// TIA Portal project "自动组装流水线" (V16)

(* hardware
DEVICE "HMI_1"  KTP700 Basic PN
   slot 0: "HMI_1"  KTP700 Basic PN  6AV2 123-2GB03-0AX0  16.0.0.0
   slot 1: "HMI_RT_1"  KTP700 Basic PN  6AV2 123-2GB03-0AX0  16.0.0.0
   slot 5: "HMI_1.IE_CP_1"  PROFINET Interface  16.0.0.0
      slot 1: "PROFINET Interface_1"  PROFINET Interface
         slot 1: "Port_1"  Port
DEVICE "S7-1200 station_1"  S7-1200 Station
   slot 0: "Rack_0"  S7-1200 Rack  Rack  V1.0
   slot 1: "PLC_1"  CPU 1214C DC/DC/Rly  6ES7 214-1HG40-0XB0  V4.4
*)

// ===== PLC "PLC_1"  CPU 1214C DC/DC/Rly =====

VAR_GLOBAL   // PLC tag table "中间变量"
   "中间变量1" AT %M0.0 : Bool;
   "中间变量2" AT %M0.1 : Bool;
   "中间变量3" AT %M0.2 : Bool;
   "中间变量4" AT %M0.3 : Bool;
   "中间变量5" AT %M0.4 : Bool;
   "中间变量6" AT %M0.5 : Bool;
   "中间变量7" AT %M0.6 : Bool;
   "中间变量8" AT %M0.7 : Bool;
   "中间变量9" AT %M1.0 : Bool;
   "中间变量10" AT %M1.1 : Bool;
   "中间变量11" AT %M1.2 : Bool;
   "中间变量12" AT %M1.3 : Bool;
   "中间变量13" AT %M1.4 : Bool;
   "中间变量14" AT %M1.5 : Bool;
   "启动" AT %M1.6 : Bool;
   "停止(1)" AT %M1.7 : Bool;
   "复位(1)" AT %M2.0 : Bool;
   "启动标志1" AT %M2.1 : Bool;
   "推杆标志1" AT %M2.2 : Bool;
   "推杆标志2" AT %M2.3 : Bool;
   "推杆收1" AT %M2.4 : Bool;
   "推杆收2" AT %M2.5 : Bool;
   "上下准备" AT %M2.6 : Bool;
   "吸附准备" AT %M2.7 : Bool;
   "吸附过程" AT %M3.0 : Bool;
   "前后准备" AT %M3.1 : Bool;
   "准备下降" AT %M3.2 : Bool;
   "断开吸附" AT %M3.3 : Bool;
   "x轴复位" AT %M3.4 : Bool;
   "皮带1状态" AT %M3.5 : Bool;
   "皮带2状态" AT %M3.6 : Bool;
   "皮带启动1" AT %M3.7 : Bool;
   "皮带启动2" AT %M4.0 : Bool;
   "上升2准备" AT %M4.1 : Bool;
   "上升2复位" AT %M4.2 : Bool;
END_VAR

VAR_GLOBAL   // PLC tag table "io表"
   "传感器9" AT %I0.0 : Bool;
   "传感器8" AT %I0.1 : Bool;
   "传感器7" AT %I0.2 : Bool;
   "传感器1" AT %I0.3 : Bool;
   "传感器2" AT %I0.4 : Bool;
   "传感器3" AT %I0.5 : Bool;
   "传感器4" AT %I0.6 : Bool;
   "传感器5" AT %I0.7 : Bool;
   "传感器6" AT %I1.0 : Bool;
   "传感器10" AT %I1.1 : Bool;
   "开始" AT %I1.2 : Bool;
   "复位" AT %I1.3 : Bool;
   "停止" AT %I1.4 : Bool;
   "紧急停止" AT %I1.5 : Bool;
   "1挡" AT %I1.6 : Bool;
   "FACTORY I/O (Running)" AT %I1.7 : Bool;
   "前后" AT %Q0.0 : Bool;
   "上下" AT %Q0.1 : Bool;
   "吸取" AT %Q0.2 : Bool;
   "皮带1" AT %Q0.3 : Bool;
   "推上盖" AT %Q0.4 : Bool;
   "上升1" AT %Q0.5 : Bool;
   "皮带2" AT %Q0.6 : Bool;
   "推下盖" AT %Q0.7 : Bool;
   "上升2" AT %Q1.0 : Bool;
   "绿灯" AT %Q1.1 : Bool;
   "黄灯" AT %Q1.2 : Bool;
   "红灯" AT %Q1.3 : Bool;
   "显示屏" AT %QD30 : DInt;
END_VAR

DATA_BLOCK "主程序"   // DB13
{ S7_Optimized_Access := 'TRUE' }
VERSION : 0.1
   VAR
      急停 : Bool := true;
      模式 : Int;
      "运行/停止" : Bool;
   END_VAR
BEGIN
END_DATA_BLOCK

// folder: 01-自动运行组装

DATA_BLOCK "自动运行组装_DB"   // DB14
{ S7_Optimized_Access := 'TRUE' }
VERSION : 0.1
// stored: InstanceOfName 自动运行组装
"自动运行组装"
BEGIN
END_DATA_BLOCK

// folder: 02-系统停止组块

DATA_BLOCK "系统停止组块_DB"   // DB2
{ S7_Optimized_Access := 'TRUE' }
VERSION : 0.1
// stored: InstanceOfName 系统停止组块
"系统停止组块"
BEGIN
END_DATA_BLOCK

// folder: System blocks/Program resources

DATA_BLOCK "IEC_Timer_0_DB_11"   // DB12
{ S7_Optimized_Access := 'TRUE' }
AUTHOR : Simatic
FAMILY : IEC
NAME : IEC_TMR
VERSION : 1.0
// stored: InstanceOfName IEC_TIMER
"IEC_TIMER"
BEGIN
END_DATA_BLOCK

// folder: (top level)

FUNCTION "MHJ-PLC-Lab-Function-S71200" : Void   // FC9000, SCL
{ S7_Optimized_Access := 'TRUE' }
VERSION : 0.1
   VAR_TEMP
      rdTimeReturn : Int;
      outputTime : DTL;
      SyncVal : Byte;
      forVal : Int;
      forVal_2 : Int;
      Value : Byte;
   END_VAR
   VAR CONSTANT
      CompVal : Byte := 16#34;
      Value_01 : Byte := 16#11;
      Value_01_DW : DWord := 16#A165_D992;
      Value_02_DW : DWord := 16#58BE_4401;
   END_VAR
BEGIN

   #Value:=PEEK(area := 16#82,
        dbNumber := 0,
        byteOffset := 511);
   #Value := #Value + 1;

   POKE(area := 16#82,
        dbNumber := 0,
        byteOffset := 511,
        value := #Value);

   POKE(area:=16#81,
        dbNumber:=0,
        byteOffset:=1016,
        value:=#Value_01_DW);
   POKE(area := 16#81,
        dbNumber := 0,
        byteOffset := 1020,
        value := #Value_02_DW);

   POKE(area := 16#81,
        dbNumber := 0,
        byteOffset := 511,
        value := B#16#00);

   FOR #forVal := 0 TO 120 DO
       FOR #forVal_2:=0 TO 10 DO
           #rdTimeReturn:=RD_SYS_T(#outputTime);
           #rdTimeReturn := WR_SYS_T(#outputTime);
           #rdTimeReturn := RD_SYS_T(#outputTime);
           #rdTimeReturn := WR_SYS_T(#outputTime);
       END_FOR;
       #SyncVal:= PEEK(area := 16#81,
                      dbNumber := 0,
                      byteOffset := 511);
       IF #SyncVal = #CompVal THEN
          GOTO M_1;
       END_IF;
   END_FOR;
   RETURN;

   M_1:
   POKE(area := 16#81,
        dbNumber := 0,
        byteOffset := 511,
        value := B#16#0);
END_FUNCTION

ORGANIZATION_BLOCK "Main"   // OB1, LAD, ProgramCycle
TITLE = "Main Program Sweep (Cycle)"
{ S7_Optimized_Access := 'TRUE' }
VERSION : 0.1
   VAR_INPUT
      Initial_Call : Bool;   // Initial call of this OB
      Remanence : Bool;   // =True, if remanent data are available
   END_VAR
   VAR_TEMP   // added for the SCL form of the ladder/FBD networks
      _w1 : Bool;
      _w2 : Bool;
   END_VAR
BEGIN

REGION Network 1
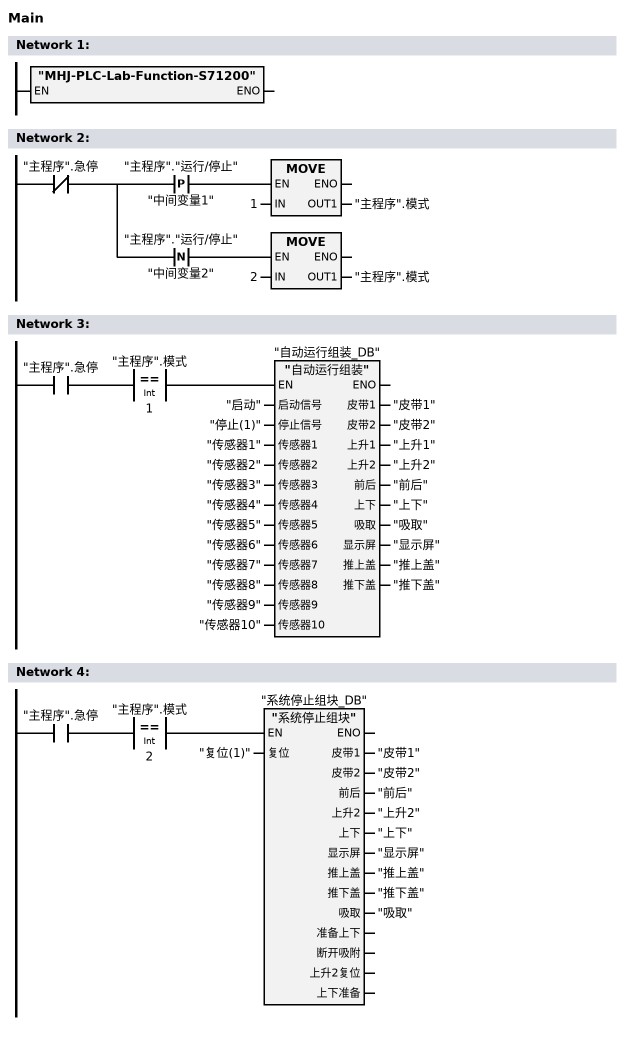
   RUNG wire#powerrail
      "MHJ-PLC-Lab-Function-S71200"()
   END_RUNG
   // the same network as SCL:
   "MHJ-PLC-Lab-Function-S71200"();
END_REGION

REGION Network 2
   RUNG wire#powerrail
      I_Contact( "主程序".急停 )
      wire#w1
      P_Contact(operand := "主程序"."运行/停止", bit := "中间变量1")
      Move(in := 1, out1 => "主程序".模式)
   END_RUNG
   RUNG wire#w1
      N_Contact(operand := "主程序"."运行/停止", bit := "中间变量2")
      Move(in := 2, out1 => "主程序".模式)
   END_RUNG
   // the same network as SCL:
   #_w1 := NOT "主程序".急停 AND "主程序"."运行/停止" AND NOT "中间变量1";   // rising edge of "主程序"."运行/停止"
   "中间变量1" := "主程序"."运行/停止";
   IF #_w1 THEN "主程序".模式 := 1; END_IF;
   #_w2 := NOT "主程序".急停 AND NOT "主程序"."运行/停止" AND "中间变量2";   // falling edge of "主程序"."运行/停止"
   "中间变量2" := "主程序"."运行/停止";
   IF #_w2 THEN "主程序".模式 := 2; END_IF;
END_REGION

REGION Network 3
   RUNG wire#powerrail
      Contact( "主程序".急停 )
      { S7_Templates := "SrcType := Int" } EQ_Contact(in1 := "主程序".模式, in2 := 1)
      "自动运行组装_DB"(启动信号 := "启动", 停止信号 := "停止(1)", 传感器1 := "传感器1", 传感器2 := "传感器2", 传感器3 := "传感器3", 传感器4 := "传感器4", 传感器5 := "传感器5", 传感器6 := "传感器6", 传感器7 := "传感器7", 传感器8 := "传感器8", 传感器9 := "传感器9", 传感器10 := "传感器10", 皮带1 => "皮带1", 皮带2 => "皮带2", 上升1 => "上升1", 上升2 => "上升2", 前后 => "前后", 上下 => "上下", 吸取 => "吸取", 显示屏 => "显示屏", 推上盖 => "推上盖", 推下盖 => "推下盖")
   END_RUNG
   // the same network as SCL:
   IF "主程序".急停 AND ("主程序".模式 = 1) THEN
       "自动运行组装_DB"(启动信号 := "启动",   // "自动运行组装"
                   停止信号 := "停止(1)",
                   传感器1 := "传感器1",
                   传感器2 := "传感器2",
                   传感器3 := "传感器3",
                   传感器4 := "传感器4",
                   传感器5 := "传感器5",
                   传感器6 := "传感器6",
                   传感器7 := "传感器7",
                   传感器8 := "传感器8",
                   传感器9 := "传感器9",
                   传感器10 := "传感器10",
                   皮带1 => "皮带1",
                   皮带2 => "皮带2",
                   上升1 => "上升1",
                   上升2 => "上升2",
                   前后 => "前后",
                   上下 => "上下",
                   吸取 => "吸取",
                   显示屏 => "显示屏",
                   推上盖 => "推上盖",
                   推下盖 => "推下盖");
   END_IF;
END_REGION

REGION Network 4
   RUNG wire#powerrail
      Contact( "主程序".急停 )
      { S7_Templates := "SrcType := Int" } EQ_Contact(in1 := "主程序".模式, in2 := 2)
      "系统停止组块_DB"(复位 := "复位(1)", 皮带1 => "皮带1", 皮带2 => "皮带2", 前后 => "前后", 上升2 => "上升2", 上下 => "上下", 显示屏 => "显示屏", 推上盖 => "推上盖", 推下盖 => "推下盖", 吸取 => "吸取", 准备上下 =>, 断开吸附 =>, 上升2复位 =>, 上下准备 =>)
   END_RUNG
   // the same network as SCL:
   IF "主程序".急停 AND ("主程序".模式 = 2) THEN
       "系统停止组块_DB"(复位 := "复位(1)",   // "系统停止组块"
                   皮带1 => "皮带1",
                   皮带2 => "皮带2",
                   前后 => "前后",
                   上升2 => "上升2",
                   上下 => "上下",
                   显示屏 => "显示屏",
                   推上盖 => "推上盖",
                   推下盖 => "推下盖",
                   吸取 => "吸取");
   END_IF;
END_REGION
END_ORGANIZATION_BLOCK

// folder: 01-自动运行组装

FUNCTION_BLOCK "自动运行组装"   // FB1, LAD
{ S7_Optimized_Access := 'TRUE' }
VERSION : 0.1
   VAR_INPUT
      启动信号 : Bool;
      停止信号 : Bool;
      传感器1 : Bool;
      传感器2 : Bool;
      传感器3 : Bool;
      传感器4 : Bool;
      传感器5 : Bool;
      传感器6 : Bool;
      传感器7 : Bool;
      传感器8 : Bool;
      传感器9 : Bool;
      传感器10 : Bool;
   END_VAR
   VAR_OUTPUT
      皮带1 : Bool;
      皮带2 : Bool;
      上升1 : Bool;
      上升2 : Bool;
      前后 : Bool;
      上下 : Bool;
      吸取 : Bool;
      显示屏 : DInt;
      推上盖 : Bool;
      推下盖 : Bool;
   END_VAR
   VAR
      启动标志 : Bool;
      皮带启动1 : Bool;
      皮带启动2 : Bool;
      皮带状态1 : Bool;
      皮带状态2 : Bool;
      推杆标志1 : Bool;
      推杆标志2 : Bool;
      推上收 : Bool;
      推下收 : Bool;
      上下准备 : Bool;
      吸附准备 : Bool;
      中间变量1 : Bool;
      中间变量2 : Bool;
      吸附过程 : Bool;
      前后准备 : Bool;
      准备上下 : Bool;
      断开吸附 : Bool;
      x轴复位 : Bool;
      上升2准备 : Bool;
      上升2复位 : Bool;
      IEC_Timer_0_Instance : TON_TIME;
      IEC_Timer_0_Instance_1 : TON_TIME;
      IEC_Timer_0_Instance_2 : TON_TIME;
      IEC_Timer_0_Instance_3 : TON_TIME;
      IEC_Timer_0_Instance_4 : TON_TIME;
      IEC_Timer_0_Instance_5 : TON_TIME;
      IEC_Timer_0_Instance_6 : TON_TIME;
      IEC_Timer_0_Instance_7 : TON_TIME;
      IEC_Timer_0_Instance_8 : TON_TIME;
      IEC_Timer_0_Instance_9 : TON_TIME;
      IEC_Timer_0_Instance_10 : TON_TIME;
      IEC_Timer_0_Instance_11 : TON_TIME;
   END_VAR
   VAR_TEMP   // added for the SCL form of the ladder/FBD networks
      _w1 : Bool;
      _w2 : Bool;
   END_VAR
BEGIN

REGION Network 1: 按下开关
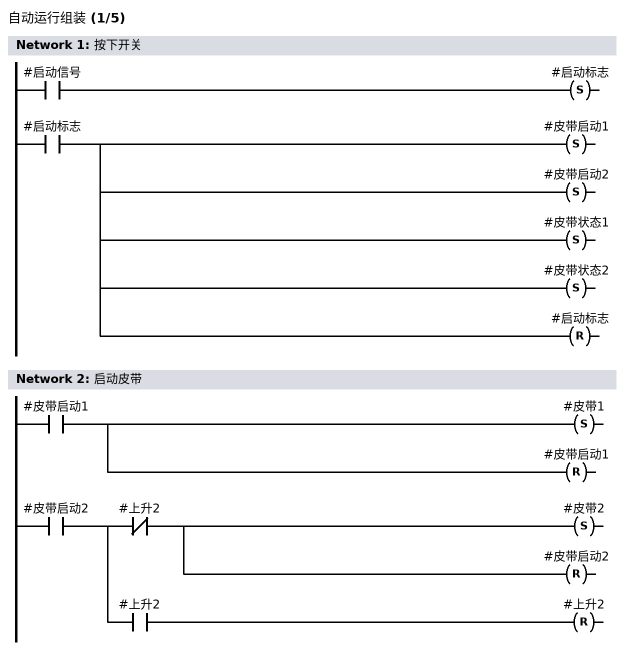
   RUNG wire#powerrail
      Contact( #启动信号 )
      S_Coil( #启动标志 )
   END_RUNG
   RUNG wire#powerrail
      Contact( #启动标志 )
      wire#w1
      S_Coil( #皮带启动1 )
   END_RUNG
   RUNG wire#w1
      S_Coil( #皮带启动2 )
   END_RUNG
   RUNG wire#w1
      S_Coil( #皮带状态1 )
   END_RUNG
   RUNG wire#w1
      S_Coil( #皮带状态2 )
   END_RUNG
   RUNG wire#w1
      R_Coil( #启动标志 )
   END_RUNG
   // the same network as SCL:
   IF #启动信号 THEN #启动标志 := TRUE; END_IF;
   IF #启动标志 THEN
       #皮带启动1 := TRUE;
       #皮带启动2 := TRUE;
       #皮带状态1 := TRUE;
       #皮带状态2 := TRUE;
       #启动标志 := FALSE;
   END_IF;
END_REGION

REGION Network 2: 启动皮带
   RUNG wire#powerrail
      Contact( #皮带启动1 )
      wire#w1
      S_Coil( #皮带1 )
   END_RUNG
   RUNG wire#w1
      R_Coil( #皮带启动1 )
   END_RUNG
   RUNG wire#powerrail
      Contact( #皮带启动2 )
      wire#w2
      I_Contact( #上升2 )
      wire#w3
      S_Coil( #皮带2 )
   END_RUNG
   RUNG wire#w3
      R_Coil( #皮带启动2 )
   END_RUNG
   RUNG wire#w2
      Contact( #上升2 )
      R_Coil( #上升2 )
   END_RUNG
   // the same network as SCL:
   IF #皮带启动1 THEN
       #皮带1 := TRUE;
       #皮带启动1 := FALSE;
   END_IF;
   IF #皮带启动2 AND NOT #上升2 THEN #皮带2 := TRUE; END_IF;
   #_w1 := #皮带启动2;
   IF #皮带启动2 AND NOT #上升2 THEN #皮带启动2 := FALSE; END_IF;
   IF #_w1 AND #上升2 THEN #上升2 := FALSE; END_IF;
END_REGION

REGION Network 3: 传感器感应到，然后停止
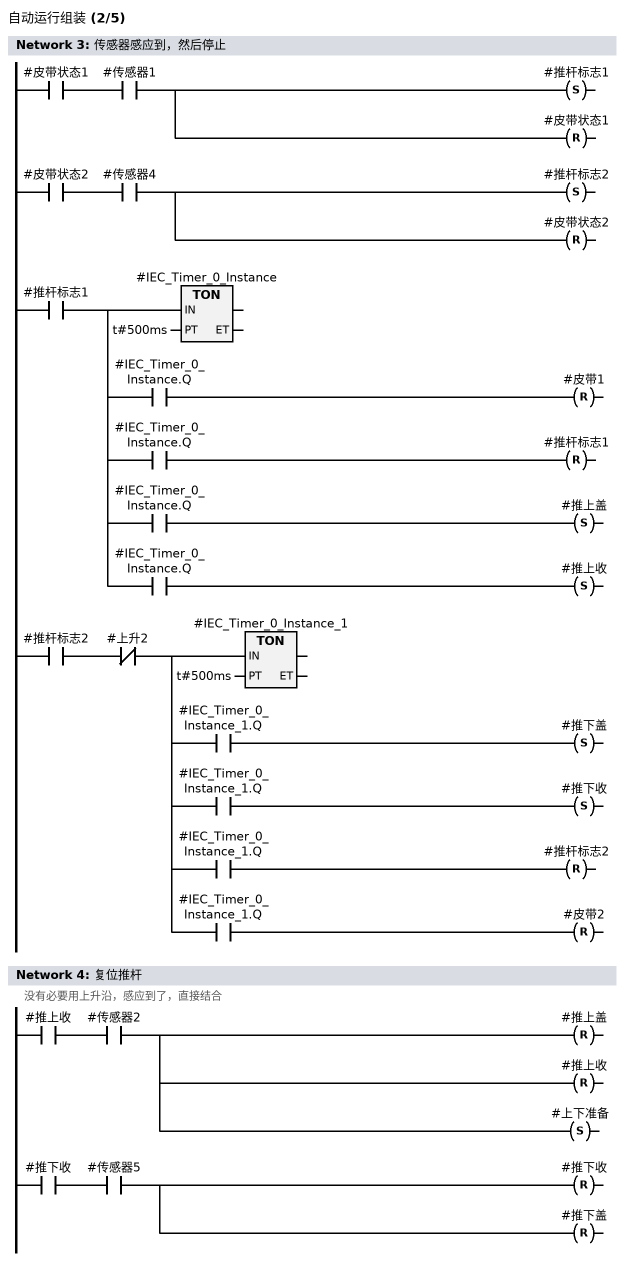
   IF #皮带状态1 AND #传感器1 THEN
       #推杆标志1 := TRUE;
       #皮带状态1 := FALSE;
   END_IF;
   IF #皮带状态2 AND #传感器4 THEN
       #推杆标志2 := TRUE;
       #皮带状态2 := FALSE;
   END_IF;
   #IEC_Timer_0_Instance(IN := #推杆标志1, PT := t#500ms);   // TON
   IF #推杆标志1 AND #IEC_Timer_0_Instance.Q THEN #皮带1 := FALSE; END_IF;
   #_w1 := #推杆标志1;
   IF #推杆标志1 AND #IEC_Timer_0_Instance.Q THEN #推杆标志1 := FALSE; END_IF;
   IF #_w1 AND #IEC_Timer_0_Instance.Q THEN
       #推上盖 := TRUE;
       #推上收 := TRUE;
   END_IF;
   #_w2 := #推杆标志2 AND NOT #上升2;
   #IEC_Timer_0_Instance_1(IN := #_w2, PT := t#500ms);   // TON
   IF #_w2 AND #IEC_Timer_0_Instance_1.Q THEN
       #推下盖 := TRUE;
       #推下收 := TRUE;
       #推杆标志2 := FALSE;
       #皮带2 := FALSE;
   END_IF;
END_REGION

REGION Network 4: 复位推杆
   // 没有必要用上升沿，感应到了，直接结合
   RUNG wire#powerrail
      Contact( #推上收 )
      Contact( #传感器2 )
      wire#w1
      R_Coil( #推上盖 )
   END_RUNG
   RUNG wire#w1
      R_Coil( #推上收 )
   END_RUNG
   RUNG wire#w1
      S_Coil( #上下准备 )
   END_RUNG
   RUNG wire#powerrail
      Contact( #推下收 )
      Contact( #传感器5 )
      wire#w2
      R_Coil( #推下收 )
   END_RUNG
   RUNG wire#w2
      R_Coil( #推下盖 )
   END_RUNG
   // the same network as SCL:
   IF #推上收 AND #传感器2 THEN #推上盖 := FALSE; END_IF;
   #_w1 := #推上收 AND #传感器2;
   IF #_w1 THEN
       #推上收 := FALSE;
       #上下准备 := TRUE;
   END_IF;
   #_w2 := #推下收 AND #传感器5;
   IF #_w2 THEN
       #推下收 := FALSE;
       #推下盖 := FALSE;
   END_IF;
END_REGION

REGION Network 5: 准备吸附
   // 利用传感器2来判断是否推到位
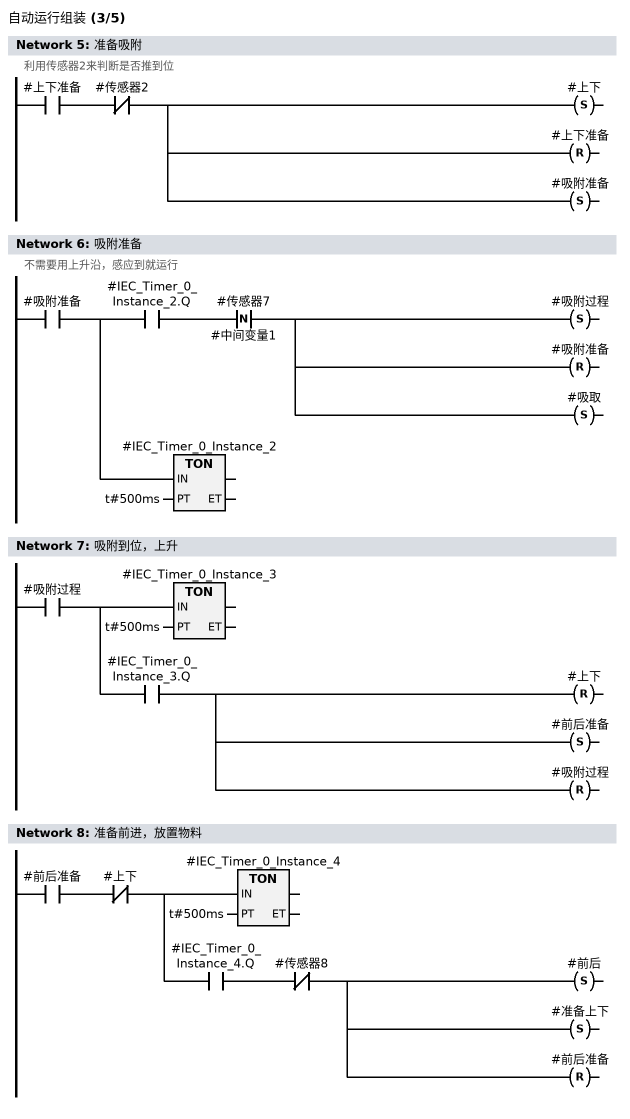
   RUNG wire#powerrail
      Contact( #上下准备 )
      I_Contact( #传感器2 )
      wire#w1
      S_Coil( #上下 )
   END_RUNG
   RUNG wire#w1
      R_Coil( #上下准备 )
   END_RUNG
   RUNG wire#w1
      S_Coil( #吸附准备 )
   END_RUNG
   // the same network as SCL:
   IF #上下准备 AND NOT #传感器2 THEN #上下 := TRUE; END_IF;
   #_w1 := #上下准备 AND NOT #传感器2;
   IF #_w1 THEN
       #上下准备 := FALSE;
       #吸附准备 := TRUE;
   END_IF;
END_REGION

REGION Network 6: 吸附准备
   // 不需要用上升沿，感应到就运行
   #_w1 := #吸附准备 AND #IEC_Timer_0_Instance_2.Q AND NOT #传感器7 AND #中间变量1;   // falling edge of #传感器7
   #中间变量1 := #传感器7;
   IF #_w1 THEN #吸附过程 := TRUE; END_IF;
   #_w2 := #吸附准备;
   IF #_w1 THEN
       #吸附准备 := FALSE;
       #吸取 := TRUE;
   END_IF;
   #IEC_Timer_0_Instance_2(IN := #_w2, PT := t#500ms);   // TON
END_REGION

REGION Network 7: 吸附到位，上升
   #IEC_Timer_0_Instance_3(IN := #吸附过程, PT := t#500ms);   // TON
   IF #吸附过程 AND #IEC_Timer_0_Instance_3.Q THEN
       #上下 := FALSE;
       #前后准备 := TRUE;
       #吸附过程 := FALSE;
   END_IF;
END_REGION

REGION Network 8: 准备前进，放置物料
   #_w1 := #前后准备 AND NOT #上下;
   #IEC_Timer_0_Instance_4(IN := #_w1, PT := t#500ms);   // TON
   IF #_w1 AND #IEC_Timer_0_Instance_4.Q AND NOT #传感器8 THEN
       #前后 := TRUE;
       #准备上下 := TRUE;
       #前后准备 := FALSE;
   END_IF;
END_REGION

REGION Network 9
   // 利用传感器不运动的时候，表示为0
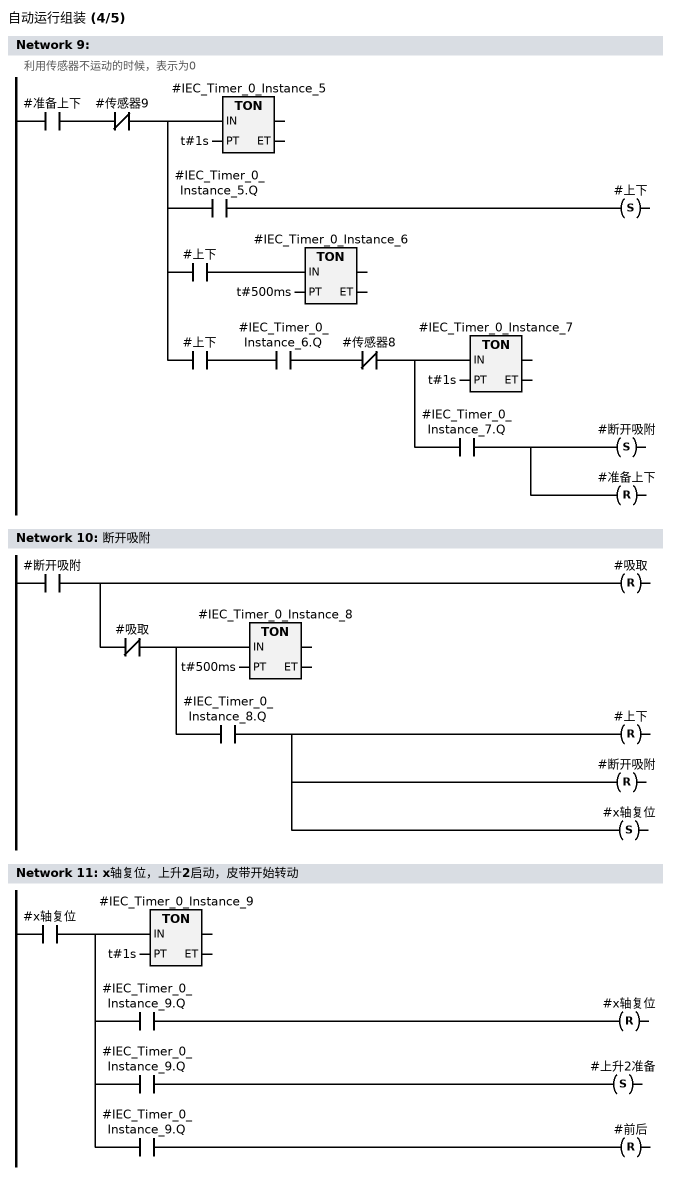
   #_w1 := #准备上下 AND NOT #传感器9;
   #IEC_Timer_0_Instance_5(IN := #_w1, PT := t#1s);   // TON
   IF #_w1 AND #IEC_Timer_0_Instance_5.Q THEN #上下 := TRUE; END_IF;
   #IEC_Timer_0_Instance_6(IN := #_w1 AND #上下, PT := t#500ms);   // TON
   #_w2 := #_w1 AND #上下 AND #IEC_Timer_0_Instance_6.Q AND NOT #传感器8;
   #IEC_Timer_0_Instance_7(IN := #_w2, PT := t#1s);   // TON
   IF #_w2 AND #IEC_Timer_0_Instance_7.Q THEN
       #断开吸附 := TRUE;
       #准备上下 := FALSE;
   END_IF;
END_REGION

REGION Network 10: 断开吸附
   IF #断开吸附 THEN #吸取 := FALSE; END_IF;
   #_w1 := #断开吸附 AND NOT #吸取;
   #IEC_Timer_0_Instance_8(IN := #_w1, PT := t#500ms);   // TON
   IF #_w1 AND #IEC_Timer_0_Instance_8.Q THEN
       #上下 := FALSE;
       #断开吸附 := FALSE;
       #x轴复位 := TRUE;
   END_IF;
END_REGION

REGION Network 11: x轴复位，上升2启动，皮带开始转动
   #IEC_Timer_0_Instance_9(IN := #x轴复位, PT := t#1s);   // TON
   #_w1 := #x轴复位;
   IF #x轴复位 AND #IEC_Timer_0_Instance_9.Q THEN #x轴复位 := FALSE; END_IF;
   IF #_w1 AND #IEC_Timer_0_Instance_9.Q THEN
       #上升2准备 := TRUE;
       #前后 := FALSE;
   END_IF;
END_REGION

REGION Network 12: 准备循环，计数
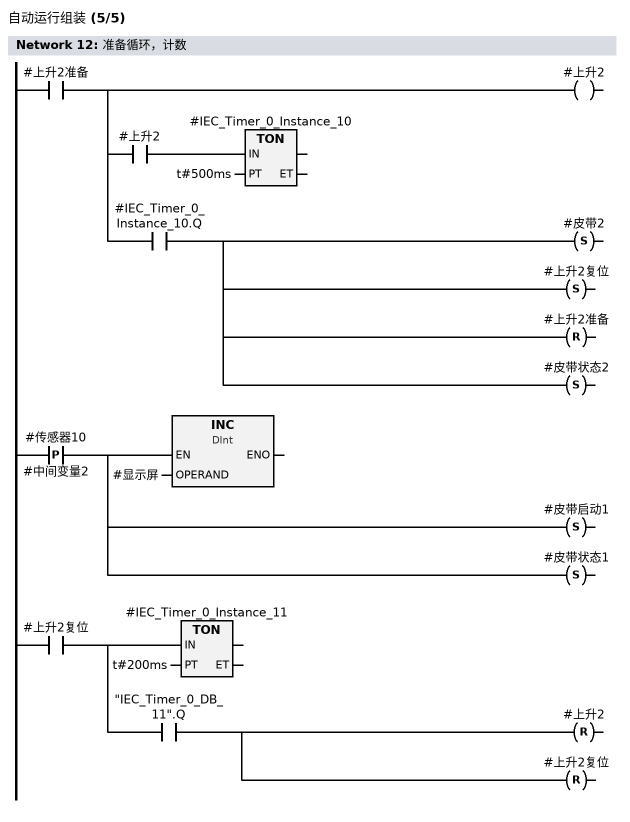
   #上升2 := #上升2准备;
   #IEC_Timer_0_Instance_10(IN := #上升2准备 AND #上升2, PT := t#500ms);   // TON
   IF #上升2准备 AND #IEC_Timer_0_Instance_10.Q THEN
       #皮带2 := TRUE;
       #上升2复位 := TRUE;
   END_IF;
   #_w1 := #上升2准备 AND #IEC_Timer_0_Instance_10.Q;
   IF #_w1 THEN
       #上升2准备 := FALSE;
       #皮带状态2 := TRUE;
   END_IF;
   #_w2 := #传感器10 AND NOT #中间变量2;   // rising edge of #传感器10
   #中间变量2 := #传感器10;
   IF #_w2 THEN
       #显示屏 := #显示屏 + 1;
       #皮带启动1 := TRUE;
       #皮带状态1 := TRUE;
   END_IF;
   #IEC_Timer_0_Instance_11(IN := #上升2复位, PT := t#200ms);   // TON
   IF #上升2复位 AND "IEC_Timer_0_DB_11".Q THEN
       #上升2 := FALSE;
       #上升2复位 := FALSE;
   END_IF;
END_REGION
END_FUNCTION_BLOCK

// folder: 02-系统停止组块

FUNCTION_BLOCK "系统停止组块"   // FB2, LAD
{ S7_Optimized_Access := 'TRUE' }
VERSION : 0.1
   VAR_INPUT
      复位 : Bool;
   END_VAR
   VAR_OUTPUT
      皮带1 : Bool;
      皮带2 : Bool;
      前后 : Bool;
      上升2 : Bool;
      上下 : Bool;
      显示屏 : Int;
      推上盖 : Bool;
      推下盖 : Bool;
      吸取 : Bool;
      准备上下 : Bool;
      断开吸附 : Bool;
      上升2复位 : Bool;
      上下准备 : Bool;
   END_VAR
BEGIN

REGION Network 1: 初始化
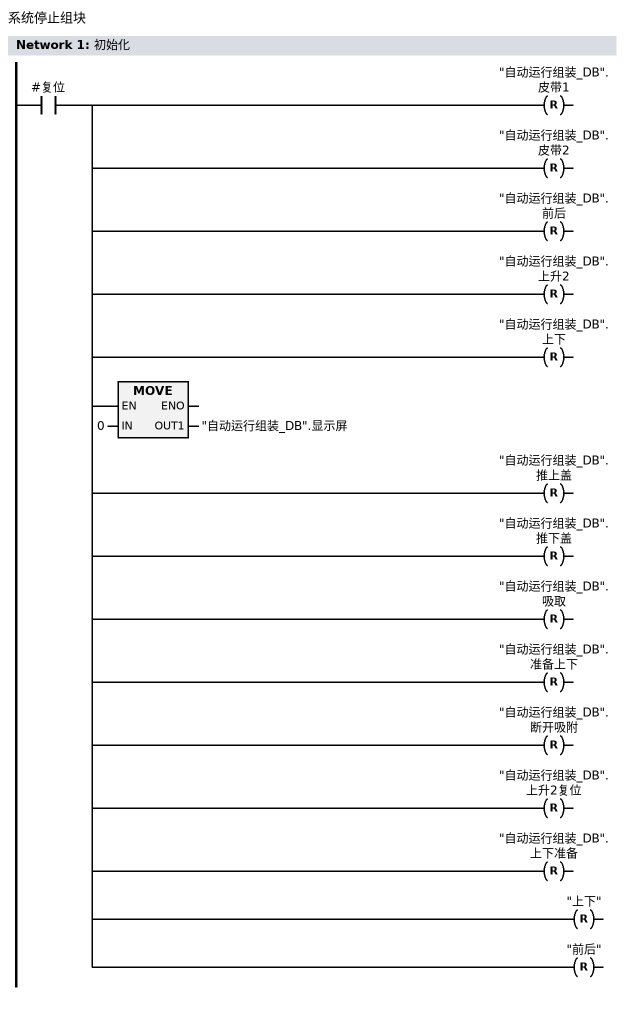
   RUNG wire#powerrail
      Contact( #复位 )
      wire#w1
      R_Coil( "自动运行组装_DB".皮带1 )
   END_RUNG
   RUNG wire#w1
      R_Coil( "自动运行组装_DB".皮带2 )
   END_RUNG
   RUNG wire#w1
      R_Coil( "自动运行组装_DB".前后 )
   END_RUNG
   RUNG wire#w1
      R_Coil( "自动运行组装_DB".上升2 )
   END_RUNG
   RUNG wire#w1
      R_Coil( "自动运行组装_DB".上下 )
   END_RUNG
   RUNG wire#w1
      Move(in := 0, out1 => "自动运行组装_DB".显示屏)
   END_RUNG
   RUNG wire#w1
      R_Coil( "自动运行组装_DB".推上盖 )
   END_RUNG
   RUNG wire#w1
      R_Coil( "自动运行组装_DB".推下盖 )
   END_RUNG
   RUNG wire#w1
      R_Coil( "自动运行组装_DB".吸取 )
   END_RUNG
   RUNG wire#w1
      R_Coil( "自动运行组装_DB".准备上下 )
   END_RUNG
   RUNG wire#w1
      R_Coil( "自动运行组装_DB".断开吸附 )
   END_RUNG
   RUNG wire#w1
      R_Coil( "自动运行组装_DB".上升2复位 )
   END_RUNG
   RUNG wire#w1
      R_Coil( "自动运行组装_DB".上下准备 )
   END_RUNG
   RUNG wire#w1
      R_Coil( "上下" )
   END_RUNG
   RUNG wire#w1
      R_Coil( "前后" )
   END_RUNG
   // the same network as SCL:
   IF #复位 THEN
       "自动运行组装_DB".皮带1 := FALSE;
       "自动运行组装_DB".皮带2 := FALSE;
       "自动运行组装_DB".前后 := FALSE;
       "自动运行组装_DB".上升2 := FALSE;
       "自动运行组装_DB".上下 := FALSE;
       "自动运行组装_DB".显示屏 := 0;
       "自动运行组装_DB".推上盖 := FALSE;
       "自动运行组装_DB".推下盖 := FALSE;
       "自动运行组装_DB".吸取 := FALSE;
       "自动运行组装_DB".准备上下 := FALSE;
       "自动运行组装_DB".断开吸附 := FALSE;
       "自动运行组装_DB".上升2复位 := FALSE;
       "自动运行组装_DB".上下准备 := FALSE;
       "上下" := FALSE;
       "前后" := FALSE;
   END_IF;
END_REGION
END_FUNCTION_BLOCK

(* ===== HMI "HMI_RT_1" =====
system functions are stored by id; their names below are inferred from use
connection "HMI_连接_1": ETHERNET, SMART_S7_1200_OMS

HMI tags "默认变量表"
   "Tag_ScreenNumber" : UInt, internal
   "启动" : Bool = PLC 启动 AT %M1.6, 1 s
   "停止(1)" : Bool = PLC "停止(1)" AT %M1.7, 1 s
   "复位(1)" : Bool = PLC "复位(1)" AT %M2.0, 1 s
   "主程序_运行/停止" : Bool = PLC 主程序.运行/停止, 1 s
   "主程序_急停" : Bool = PLC 主程序.急停, 1 s

Template "模板_1" 800x480
   Button "退出" at 714,429 size 71x50; TextOff '退出'; PictureOff "ExitRuntime_KTP700_Basic_PN_TR"; PictureOn "ExitRuntime_KTP700_Basic_PN_TR"
      on Release: StopRuntime(0)
   Button "Template_Button" at 614,429 size 71x50; TextOff 'Text'
   Button "Template_Button_1" at 514,429 size 71x50; TextOff 'Text'
   Button "Template_Button_2" at 414,429 size 71x50; TextOff 'Text'
   Button "Template_Button_3" at 314,429 size 71x50; TextOff 'Text'
   Button "Template_Button_4" at 214,429 size 71x50; TextOff 'Text'
   Button "Template_Button_5" at 114,429 size 71x50; TextOff 'Text'
   Button "起始画面" at 14,429 size 71x50; TextOff '起始画面'; PictureOff "NavigateHome_KTP700_Basic_PN_TR"; PictureOn "NavigateHome_KTP700_Basic_PN_TR"
      on Release: ActivateScreen("根画面", 0)
   SymbolicIOField "Symbolic_IO_Field_Screen" at 93,9 size 600x33; TextOff '0'; TextOn '1'; TextList "TextList_ScreenNames"
      ProcessValue <- "Tag_ScreenNumber"
      on Change: ActivateScreenByNumber("Tag_ScreenNumber", 0)
   DateTimeField "HmiScreenItemData" at 695,25 size 105x25
   DateTimeField "HmiScreenItemData_1" at 695,0 size 105x25
   GraphicView "Logo" at 0,0 size 91x51; Picture "HMI_1 的 Logo"

screen "根画面" 800x480, template "模板_1"
   on GenerateScreen: SetTag("Tag_ScreenNumber", 1)
   Button "按钮_1" at 154,169 size 96x32; TextOff '启动'
      on Press: SetBit("启动")
      on Release: ResetBit("启动")
   Button "按钮_2" at 152,251 size 96x32; TextOff '停止'
      on Release: ResetBit("停止(1)")
      on Press: SetBit("停止(1)")
   Button "按钮_3" at 150,333 size 96x32; TextOff '复位'
      on Press: SetBit("复位(1)")
      on Release: ResetBit("复位(1)")
   Switch "开关_1" at 429,192 size 166x47; CaptionText 'Switch'; TextOff '关闭'; TextOn '运行'
      ProcessValue <- "主程序_运行/停止"
   Button "按钮_4" at 366,333 size 96x32; TextOff '急停'
      on Click: InvertBit("主程序_急停")
*)